{attribute 'qualified_only'}
VAR_GLOBAL PERSISTENT
	
	ROI_Size : TcVnRotatedRectangle;
	Calibration_Factor : LREAL;
	
END_VAR
VAR_GLOBAL
	
	Start_Camera_Sequence : BOOL;
	Trigger_Image : BOOL;
	Image_Count : UINT;
	Images_Omitted : ULINT;
	
	ImageIn				: ITcVNImage;
	ImageInGrayDisplay	: ITcVnDisplayableImage;
	ImageInRawImage		: ITcVnDisplayableImage;
	ImageInInfo 		: TcVnImageInfo;
	
END_VAR

(* stored: Version 1.1.0.1, ProductVersion 3.1.4024.12
   GVL GVL_Vision: Id {70fb6ce6-48f1-4f16-8bb5-1613b625a0d8} *)
